(* IEC 61131-3 sources: UniTest/iecUnitTest_br/Library_tests/test_assertGreaterEqual_UINT, 2 files *)

(* ---- LocalVariables.var ---- *)
VAR
    vTestCases : ARRAY[0..20] OF utTestCase; (*Definition of all test cases for this POU*)
    testRunner : utTestSuite; (*Test Suite fb instance to run the tests*)
    vRunAll : BOOL; (*Manual command to run all tests for this POU*)
    vResetAll : BOOL; (*Manual command to reset all tests for this POU*)
    vTestCase1_act : UINT; (*Test data 1 of test case 1*)
    vTestCase1_xp : UINT; (*Test data 2 of test case 1*)
    vTestCase2_act : UINT; (*Test data 1 of test case 2*)
    vTestCase2_xp : UINT; (*Test data 2 of test case 2*)
    vTestCase3_act : UINT; (*Test data 1 of test case 3*)
    vTestCase3_xp : UINT; (*Test data 2 of test case 3*)
END_VAR

(* ---- main.st ---- *)
PROGRAM _CYCLIC
    (*https://github.com/tkucic/iecUnitTest/blob/main/docs/docs/ns/Library_tests/prg/test_assertGreaterEqual_UINT.md*)
    (*Run the test cases*)
    TEST_CASE_1_SETUP();
    TEST_CASE_1_EXEC();

    TEST_CASE_2_SETUP();
    TEST_CASE_2_EXEC();

    TEST_CASE_3_SETUP();
    TEST_CASE_3_EXEC();

    (*Instantiate the test runner*)
    testRunner(
    	Id := 79,
    	Name := 'assertGreaterEqual_UINT',
        RunTests := GVL.RunAll OR vRunAll,
    	ResetTests := GVL.ResetAll OR vResetAll,
    	TestCases:=vTestCases);

    (*Report the results to the collection global*)
    GVL.Results[testRunner.Id] := testRunner.Summary;
END_PROGRAM
